FUNCTION_BLOCK BaseGripper
VAR_INPUT
END_VAR
VAR_OUTPUT
END_VAR
VAR
END_VAR

END_FUNCTION_BLOCK

(* stored: Version 1.1.0.1, ProductVersion 3.1.4024.9
   POU BaseGripper: Id {fac26416-acca-4852-af75-96dabb5316b0}, SpecialFunc None *)
